FUNCTION_BLOCK BLINK
VAR_INPUT
	TOGGLE : BOOL; // Indítja és leállítja a villogást
	ON_TIME : TIME; // Bekapcsolva töltött idő
	OFF_TIME : TIME; // Kikapcsolva töltött idő
END_VAR
VAR_OUTPUT
	LED : BOOL; // A led változó ami villogni fog
END_VAR
VAR
	clk1 :TON;
	clk2 :TON;
	i: INT;
END_VAR

clk1(PT:=ON_TIME);
clk2(PT:=OFF_TIME);
IF TOGGLE  THEN
	CASE i OF

0:
LED := TRUE;
clk1.IN := TRUE;
clk2.IN := FALSE;
IF clk1.Q THEN
i :=1;  
END_IF
1:
LED := FALSE;
clk1.IN := FALSE;
clk2.IN := TRUE;
IF clk2.Q THEN
	i := 0;
END_IF
	END_CASE
ELSE
		LED := FALSE;
		i:=0;
END_IF

END_FUNCTION_BLOCK

(* stored: Version 1.1.0.1, ProductVersion 3.1.4024.11
   POU BLINK: Id {3dd4618a-ca30-425e-b982-aab11e04e1f4}, SpecialFunc None *)
